// Automatisch erzeugter Code: NICHT EDITIEREN
FUNCTION CheckRangeUnsigned : UDINT
VAR_INPUT
	value, lower, upper: UDINT;
END_VAR

// Automatisch erzeugter Code: Es handelt sich hierbei um einen Implementierungsvorschlag.
{noflow}
IF (value < lower) THEN
	CheckRangeUnsigned := lower;
ELSIF(value > upper) THEN
	CheckRangeUnsigned := upper;
ELSE
	CheckRangeUnsigned := value;
END_IF
{flow}

END_FUNCTION

(* stored: Version 1.1.0.1, ProductVersion 3.1.4024.10
   POU CheckRangeUnsigned: Id {fb71cd9f-e948-42a8-81b5-a7b0be300722}, SpecialFunc CheckRangeUnsigned *)
